FUNCTION_BLOCK LOF
  {SET_ATTRIBUTE(OpcUa, SERVICE)}
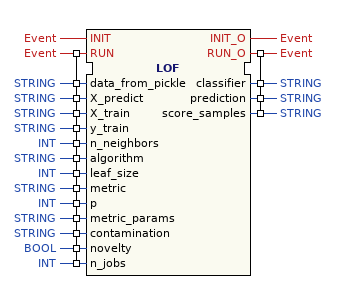
  EVENT_INPUT
    INIT;
    RUN WITH data_from_pickle, X_predict, X_train, y_train, n_neighbors, algorithm, leaf_size, metric, p, metric_params, contamination, novelty, n_jobs; {SET_ATTRIBUTE(OpcUa, Method)}
  END_EVENT
  EVENT_OUTPUT
    INIT_O;
    RUN_O WITH classifier, prediction, score_samples;
  END_EVENT
  VAR_INPUT
    data_from_pickle : STRING; {SET_ATTRIBUTE(OpcUa, Variable.RUN)}
    X_predict : STRING; {SET_ATTRIBUTE(OpcUa, Variable.RUN)}
    X_train : STRING; {SET_ATTRIBUTE(OpcUa, Variable.RUN)}
    y_train : STRING; {SET_ATTRIBUTE(OpcUa, Variable.RUN)}
    n_neighbors : INT; {SET_ATTRIBUTE(OpcUa, Variable.RUN)}
    algorithm : STRING; {SET_ATTRIBUTE(OpcUa, Variable.RUN)}
    leaf_size : INT; {SET_ATTRIBUTE(OpcUa, Variable.RUN)}
    metric : STRING; {SET_ATTRIBUTE(OpcUa, Variable.RUN)}
    p : INT; {SET_ATTRIBUTE(OpcUa, Variable.RUN)}
    metric_params : STRING; {SET_ATTRIBUTE(OpcUa, Variable.RUN)}
    contamination : STRING; {SET_ATTRIBUTE(OpcUa, Variable.RUN)}
    novelty : BOOL; {SET_ATTRIBUTE(OpcUa, Variable.RUN)}
    n_jobs : INT; {SET_ATTRIBUTE(OpcUa, Variable.RUN)}
  END_VAR
  VAR_OUTPUT
    classifier : STRING; {SET_ATTRIBUTE(OpcUa, Variable.RUN)}
    prediction : STRING; {SET_ATTRIBUTE(OpcUa, Variable.RUN)}
    score_samples : STRING; {SET_ATTRIBUTE(OpcUa, Variable.RUN)}
  END_VAR
END_FUNCTION_BLOCK
